TYPE CmpWorkStopMainLnSw :
STRUCT
	
	Framework: Framework;
	Config: CmpWorkStopMainLnSwConfig;
	Sim: CmpWorkStopMainLnSwSim;
	
	WorkReq: BOOL;
	WorkCmp: BOOL;
	PuckLnSw: PuckLnSw;
	
	DevicePresent: BOOL;
	
END_STRUCT
END_TYPE

(* stored: Version 1.1.0.1, ProductVersion 3.1.4024.6
   DUT CmpWorkStopMainLnSw: Id {84217583-e6c6-4f6c-baab-faea476a08b5} *)
